Staubli VAL3: TCPserver.pgx

program TCPserver()
  local num l_nStatus
  local num l_nBytesIn[40]
  local num l_nSuccBytes
  local pointRx p_point
  local bool erreichbar
  local bool error
begin
  // l_nBytesIn: 64 bit -> 8 byte
  // nData: 8



  while true
    logMsg("Schleife start")
    l_nStatus=sioGet(soTcpClient, l_nBytesIn)
    if l_nStatus>0
      // Write recieved bytes in data
      // Achtung bei mehr Bitlänge 24, 3 und globale Variable(nData) ändern

      if(fromBinary(l_nBytesIn,40,"8.0l",nData)!=5)
        logMsg("Empfangene Daten sind fehlerhaft",2)

      else
        logMsg("Daten über TCP/IP empfangen")
        // check if data is in limits
        // ...
        nObj = limit(nData[0],1,10)
        nOrientation = limit(nData[1],1,2)
        nX = limit(nData[2],1,750)
        nY = limit(nData[3],1,500)
        nAngle = nData[4]
        // logMsg(toString(".4",nData[0]))
        //logMsg(toString(".4",nData[1]))
        //logMsg(toString(".4",nData[3]))
        //logMsg(toString(".4",nY))
        //logMsg(toString(".4",nData[3]))
        //logMsg(toString(".4",nData[4]))


        // check if the Point is reachable
        error = false
        pEmpty.trsf.x = nX
        pEmpty.trsf.y = nY
        pEmpty.trsf.z = 10
        pEmpty.trsf.rz = nAngle
        //
        if nData[0] == 3
          while !pointToJoint(tGreiferM,jHome,pEmpty,jEmpty)
            pEmpty.trsf.rz = pEmpty.trsf.rz + 5
            nAngle = pEmpty.trsf.rz
          endWhile
        endIf


        if !pointToJoint(tGreiferM,jHome,pEmpty,jEmpty)
          pEmpty.trsf.rz = nAngle + 180


          if pointToJoint(tGreiferM,jHome,pEmpty,jEmpty)
            nAngle = nAngle + 180
           // logMsg("Punkt wird verändert")
          else
            // logMsg("Punkt nicht erreichbar")

            error = true
          endIf

        endIf


        if error == false


          // if Vereinzeln ist True
          if nData[0]==3

            bPick = false
            bVereinzeln = true
          else
            bPick = true
            bVereinzeln = false
          endIf



          bReady = false
          bNewData = true

        else
          bReady = true
          logMsg(" ****************** Punkt ist nicht erreichbar!!")

        endIf

      endIf



      // tell client that robot is ready
      wait(bReady)

      //delay(2)
      l_nStatus=sioSet(soTcpClient, 1)
    endIf
  endWhile
end
